FUNCTION_BLOCK FB_UnpackByteToBoolArray
VAR_INPUT
	inputByte : BYTE;
END_VAR
VAR_IN_OUT
    outputBits : ARRAY[0..7]OF BOOL;
END_VAR
VAR
    idx : INT;
END_VAR
//-----------------------------oldschoo1

FOR idx := 0 TO 7 
DO
outputBits[idx] := (inputByte AND SHL(1, idx)) <> 0;
END_FOR
//------------------------------------------oldschoo1

END_FUNCTION_BLOCK

(* stored: Version 1.1.0.1, ProductVersion 3.1.4024.12
   POU FB_UnpackByteToBoolArray: Id {c523551d-309a-402b-9c4e-707ae2a9da6e}, SpecialFunc None *)
